{attribute 'qualified_only'}
{attribute 'strict'}
TYPE E_Message_Grid :
(
	eNoMessage := 0,
	eTooMuchGrids := 1,
	eGridError := 2,
	eNoConnectionToBackend := 3
);
END_TYPE

(* stored: Version 1.1.0.1, ProductVersion 3.1.4024.6
   DUT E_Message_Grid: Id {3cdd75e0-2da2-40c6-9336-98ffd3b5b2eb} *)
